FUNCTION_BLOCK MotionArgument IMPLEMENTS I_LogArgument
VAR
	_Pars : REFERENCE TO ST_MotionParameters;
END_VAR

PROPERTY Parameters : REFERENCE TO ST_MotionParameters
GET
Parameters := _Pars;
END_GET
SET
_Pars REF= Parameters;
END_SET
END_PROPERTY

METHOD ToString : Logging_Helper.T_MaxString
ToString := CONCAT('Vel: ', CONCAT(TO_STRING(_Pars.Velocity), CONCAT(' Accel: ', CONCAT(TO_STRING(_Pars.Accel), CONCAT(' Decel: ', CONCAT(TO_STRING(_Pars.Decel), CONCAT(' Jerk: ',TO_STRING(_Pars.Jerk))))))));
END_METHOD

END_FUNCTION_BLOCK

(* stored: Version 1.1.0.1, ProductVersion 3.1.4026.18
   POU MotionArgument: Id {52e064b7-5081-4d35-b2ef-fdf75d75d196}, SpecialFunc None
   Property Parameters: Id {8dd60db5-ab77-49a5-b82a-1c10d97f71ab}
   Get Get: Id {73c7b1f6-6c5d-43ef-9948-7f3c32e05c54}
   Set Set: Id {37c52a50-825f-473a-9b57-63dfc3d52d38}
   Method ToString: Id {ac385968-e963-447f-9c9e-ac4174389186} *)
